FUNCTION_BLOCK EQ_Conveyor_V1
VAR_INPUT
	PS_101: BOOL; // Proximity switch
	PS_102: BOOL;
	
	STOP: BOOL;
END_VAR
VAR_OUTPUT
	M_101_CW : BOOL;
	M_101_CCW : BOOL;
	
	Alarm_1: BOOL;
	Alarm_2: BOOL;
END_VAR
VAR
	TRIG_LS_101: Tc2_Standard.R_TRIG;
	TRIG_LS_102: Tc2_Standard.R_TRIG;
	SR_M_101_CW: SR;
	SR_M_101_CCW: SR;
	TON_M101_CW: TON;
	TON_M102_CW: TON;
	
END_VAR

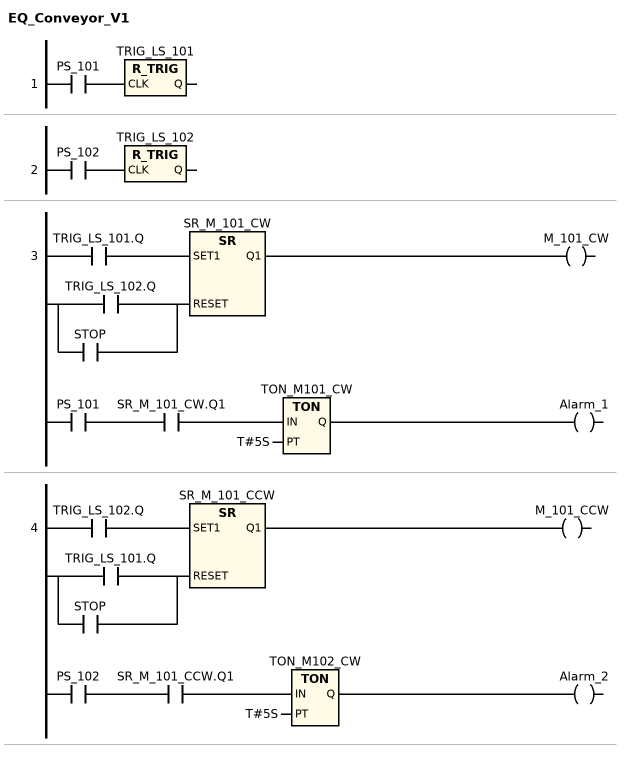
// NETWORK 1
TRIG_LS_101(CLK := PS_101); // R_TRIG

// NETWORK 2
TRIG_LS_102(CLK := PS_102); // R_TRIG

// NETWORK 3
SR_M_101_CW(SET1 := TRIG_LS_101.Q, RESET := TRIG_LS_102.Q OR STOP); // SR
M_101_CW := SR_M_101_CW.Q1;
TON_M101_CW(IN := PS_101 AND SR_M_101_CW.Q1, PT := T#5S); // TON
Alarm_1 := TON_M101_CW.Q;

// NETWORK 4
SR_M_101_CCW(SET1 := TRIG_LS_102.Q, RESET := TRIG_LS_101.Q OR STOP); // SR
M_101_CCW := SR_M_101_CCW.Q1;
TON_M102_CW(IN := PS_102 AND SR_M_101_CCW.Q1, PT := T#5S); // TON
Alarm_2 := TON_M102_CW.Q;

END_FUNCTION_BLOCK

(* stored: Version 1.1.0.1, ProductVersion 3.1.4024.13
   POU EQ_Conveyor_V1: Id {d34b433d-a8b8-45c8-ab30-28e99808cabf}, SpecialFunc None *)
